RoboDK station: estacion_practica_tablero.rdk

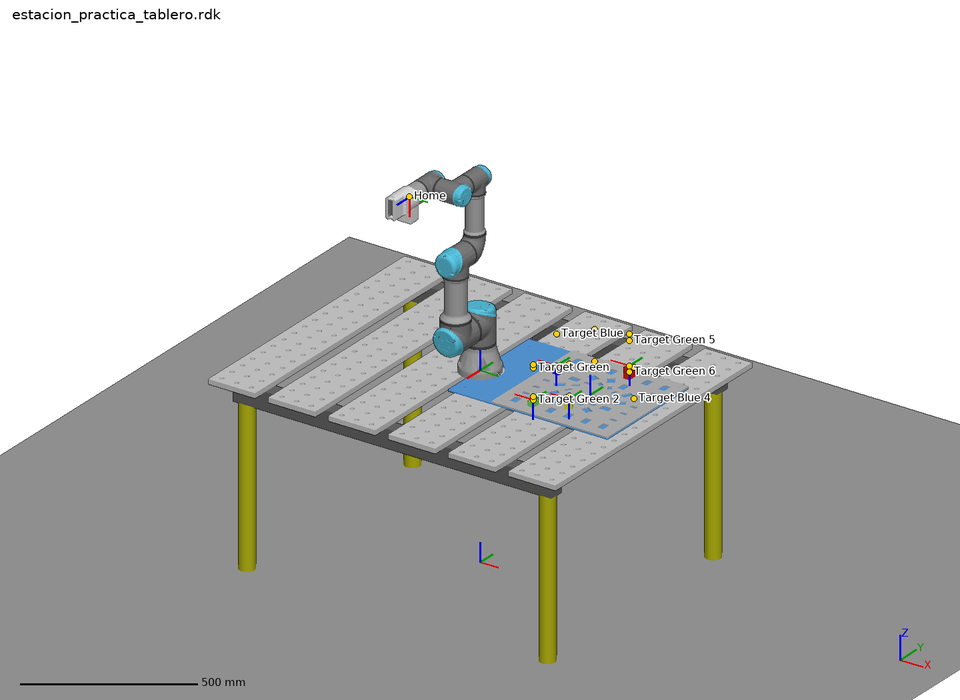
[picture v0: the station drawn from its stored meshes, robots at their saved joint values, targets as dots, program paths as lines]
Station estacion_practica_tablero (saved by RoboDK 5.6.2). Poses are relative to the parent item; angles as X-Y-Z fixed-axis rotations.
  - frame Ground at (0, 1000, 0) mm
    - object Floor at (0, 0, 0) mm, size 3000 x 3000 x 0 mm, geometry from suelo.sld
    - frame Table at (0, 0, 600) mm
      - object Table 1200x1000mm (Welding) at (0, 0, 0) mm, size 1193.8 x 965.2 x 609.6 mm, geometry from mesa.sld
      - frame Base frame at (0, 0, 0) mm
        - object _PIEZA_BaseDeTrabajo at (550, -160, 0) mm, rotated rx 90 ry 0 rz 180 deg, size 550 x 5 x 400 mm, geometry from _PIEZA_BaseDeTrabajo.STL
        - frame workframe at (350, 40, 5) mm
          - object _PIEZA_RebordeBaseDeTrabajoParaBloques at (-200, 200, 0) mm, rotated rx 90 ry 0 rz 0 deg, size 400 x 5 x 400 mm, geometry from _PIEZA_RebordeBaseDeTrabajoParaBloques.STL
          - frame Block1 at (-90, -150, 20) mm, rotated rx 180 ry 0 rz 180 deg
            - target Target Green (Cartesian target) at (0, 0, -100) mm; joints [95, -80, -112, -78, 90, 95] of UR3e
            - target Target Green 2 (Cartesian target) at (0, 0, 0) mm; joints [94.727, -92.665, -131.329, -46.005, 90, 94.727] of UR3e
            - target Target Green 5 (Cartesian target) at (-120, 300, -100) mm; joints [134.531, -116.035, -70.33, -83.635, 90, -225.469] of UR3e
            - target Target Green 6 (Cartesian target) at (-120, 300, 0) mm; joints [134.531, -123.597, -86.734, -59.669, 90, -225.469] of UR3e
            - target Target Green 3 (Cartesian target) at (0, 300, -100) mm; joints [150.172, -90.272, -102.835, -76.893, 90, -209.828] of UR3e
            - target Target Green 4 (Cartesian target) at (0, 300, 0) mm; joints [150.172, -102.012, -120.117, -47.87, 90, -209.828] of UR3e
            - object _PIEZA_Bloque20x30x20 at (10, -15, 0) mm, rotated rx 0 ry 0 rz 90 deg, size 30 x 20 x 20 mm, geometry from _PIEZA_Bloque20x30x20.STL
          - frame Block2 at (-150, 50, 30) mm, rotated rx 180 ry 0 rz 180 deg
            - target Target Blue (Cartesian target) at (0, 0, -100) mm; joints [150.921, -59.768, -121.637, -88.596, 90, 150.921] of UR3e
            - target Target Blue 2 (Cartesian target) at (0, 0, 0) mm; joints [150.921, -70.046, -145.429, -54.526, 90, 150.921] of UR3e
            - target Target Blue 3 (Cartesian target) at (-300, -50, -100) mm; joints [109.719, -142.589, -21.837, -105.573, 90, 109.719] of UR3e
            - target Target Blue 4 (Cartesian target) at (-300, -50, 0) mm; joints [109.719, -141.54, -50.998, -77.463, 90, 109.719] of UR3e
            - object _PIEZA_Bloque20x30x10 at (-10, -5, 50) mm, rotated rx 0 ry 90 rz 0 deg, size 30 x 10 x 20 mm, geometry from _PIEZA_Bloque20x30x10.STL
          - frame Block3 at (30, 150, 40) mm, rotated rx 180 ry 0 rz 180 deg
            - target Target Red (Cartesian target) at (0, 0, -100) mm; joints [134.531, -115.703, -65.44, -88.857, 90, 134.531] of UR3e
            - target Target Red 2 (Cartesian target) at (0, 0, 0) mm; joints [278.599, -58.623, 84.405, -115.782, -90, 98.599] of UR3e
            - target Target Red 3 (Cartesian target) at (29, -254, -100) mm, rotated rx 0 ry 0 rz -30 deg; joints [101.216, 180.475, 88.73, -179.206, 90, 71.216] of UR3e
            - target Target Red 4 (Cartesian target) at (29, -254, 0) mm, rotated rx 0 ry 0 rz -30 deg; joints [101.216, 156.592, 107.217, -173.809, 90, 71.216] of UR3e
            - object _PIEZA_Bloque20x30x40 at (-10, -15, 0) mm, rotated rx 90 ry 0 rz 90 deg, size 30 x 40 x 20 mm, geometry from _PIEZA_Bloque20x30x40.STL
          - frame Block4 at (1, -104, 30) mm, rotated rx 180 ry 0 rz 180 deg
            - target Target Yellow (Cartesian target) at (0, 0, -100) mm, rotated rx 0 ry 0 rz -30 deg; joints [101.216, -98.571, -91.05, -80.38, 90, 71.216] of UR3e
            - target Target Yellow 2 (Cartesian target) at (0, 0, 0) mm, rotated rx 0 ry 0 rz -30 deg; joints [101.216, -107.914, -108.495, -53.591, 90, 71.216] of UR3e
            - target Target Yellow 3 (Cartesian target) at (91, -46, -100) mm; joints [94.727, -79.169, -110.011, -80.821, 90, 94.727] of UR3e
            - target Target Yellow 4 (Cartesian target) at (91, -46, 0) mm; joints [94.727, -90.583, -129.873, -49.544, 90, 94.727] of UR3e
            - object _PIEZA_Bloque20x30x30 at (-15, -8, 30) mm, rotated rx 0 ry 90 rz -30 deg, size 30 x 30 x 20 mm, geometry from _PIEZA_Bloque20x30x30.STL
        - frame UR3e Base at (0, 0, 0) mm, rotated rx 0 ry 0 rz -90 deg
          - robot UR3e: 6 axes, payload 3 kg, reach 500 mm, repeatability 0.03 mm, weight 11 kg
              modified DH rows (alpha deg, a mm, theta deg, d mm): 0, 0, 0, 151.9; 90, 0, 180, 0; 0, 243.55, 0, 0; 0, 213.2, 0, 131.05; -90, 0, 0, 85.35; 90, 0, 180, 92.1
              joint limits [-360, -360, -360, -360, -360, -360] to [360, 360, 360, 360, 360, 360]; home [0, -90, -90, 0, 90, 0]; saved at [90, -90, 0, 0, 0, 0]
            - frame Gripper at (0, 0, 0) mm
              - robot Zimmer HRC-03 Gripper: 1 axes
                  joint limits [0] to [22]; home [0]; saved at [0]
              - target Close (joint target) at (0, 0, 130) mm; joints [12, 8.271, 64.8, -163.072, 90, -323.532] of Zimmer HRC-03 Gripper
              - target Open (joint target) at (0, 0, 130) mm; joints [0, -121.091, -92.632, -56.277, 90, -179.182] of Zimmer HRC-03 Gripper
            - tool Tool 1, TCP at (0, 0, 130) mm
    - target Home (joint target) at (-85.35, -223.15, 1208.65) mm, rotated rx 0 ry 90 rz -90 deg; joints [90, -90, 0, 0, 0, 0] of UR3e
